PROGRAM MAIN
VAR
	ManualControl_0: ManualControl;
	AutomaticControl_0: AutomaticControl;
END_VAR

// Initially it goes to position (0,0,0,0) and initializes motors by Initialize PRG.
// There is Safety PRG that keeps checking if motors are out of bounds.
// Motors are instantiated as global vars to retain their properties.
// CountCurrentPosition PRG is the only place where we count position using the sensors.
// POPRAVI SMERI: RestorePreviousAutomaticState is a FB that gets execture cyclic until all the directions are set to previous positions.
// AutomaticControl FB remembers which recipe is being executed and recipe remembers its state.

// TODO:
// delay...
VAR // added by the converter: edge detectors and wires of the graphical bodies
    _w1, _w2 : BOOL;
    _rt1, _rt2 : R_TRIG;
    _ft1 : F_TRIG;
END_VAR

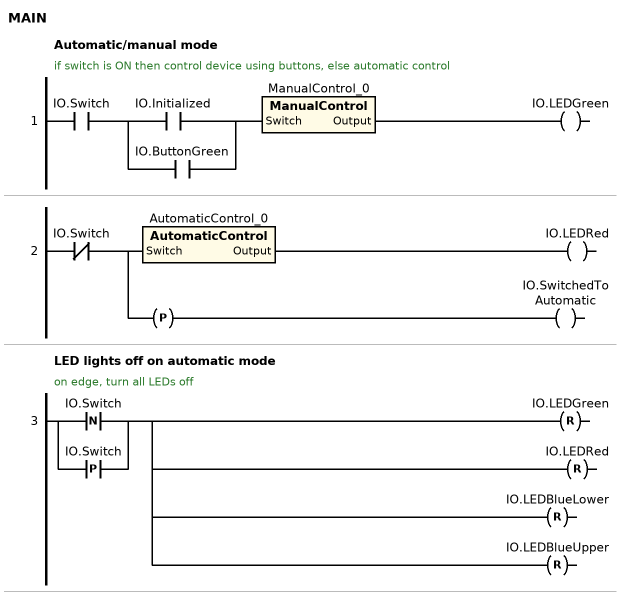
// NETWORK 1: Automatic/manual mode
// if switch is ON then control device using buttons, else automatic control
ManualControl_0(Switch := IO.Switch AND IO.Initialized OR IO.Switch AND IO.ButtonGreen); // ManualControl
IO.LEDGreen := ManualControl_0.Output;

// NETWORK 2
_w1 := NOT IO.Switch;
AutomaticControl_0(Switch := _w1); // AutomaticControl
IO.LEDRed := AutomaticControl_0.Output;
_rt1(CLK := _w1);
IO.SwitchedToAutomatic := _rt1.Q;

// NETWORK 3: LED lights off on automatic mode
// on edge, turn all LEDs off
_ft1(CLK := IO.Switch);
_rt2(CLK := IO.Switch);
_w2 := _ft1.Q OR _rt2.Q;
IO.LEDGreen R= _w2;
IO.LEDRed R= _w2;
IO.LEDBlueLower R= _w2;
IO.LEDBlueUpper R= _w2;

END_PROGRAM

(* stored: Version 1.1.0.1, ProductVersion 3.1.4024.13
   POU MAIN: Id {ca0d1193-1c86-427a-9c71-41bf6bccd822}, SpecialFunc None *)
